// TIA Portal project "Project2" (V16)

(* hardware
DEVICE "S7-1200 station_1"  S7-1200 Station
   slot 0: "Rack_0"  S7-1200 Rack  Rack  V1.0
   slot 1: "PLC_1"  CPU 1212C AC/DC/Rly  6ES7 212-1BE40-0XB0  V4.4
*)

// ===== PLC "PLC_1"  CPU 1212C AC/DC/Rly =====

VAR_GLOBAL   // PLC tag table "Default tag table"
   "START" AT %I0.1 : Bool;
   "STOP" AT %I0.2 : Bool;
   "MOTOR1" AT %Q0.0 : Bool;
   "MOTOR2" AT %Q0.1 : Bool;
   "MOTOR3" AT %Q0.2 : Bool;
   "Tag_1" AT %M0.0 : Bool;
   "Tag_2" AT %M0.1 : Bool;
   "Tag_3" AT %M0.2 : Bool;
   "Tag_4" AT %M0.3 : Bool;
END_VAR

// folder: System blocks/Program resources

DATA_BLOCK "TIMER1"   // DB1
{ S7_Optimized_Access := 'TRUE' }
AUTHOR : Simatic
FAMILY : IEC
NAME : IEC_TMR
VERSION : 1.0
// stored: InstanceOfName IEC_TIMER
"IEC_TIMER"
BEGIN
END_DATA_BLOCK

DATA_BLOCK "TIMER2"   // DB2
{ S7_Optimized_Access := 'TRUE' }
AUTHOR : Simatic
FAMILY : IEC
NAME : IEC_TMR
VERSION : 1.0
// stored: InstanceOfName IEC_TIMER
"IEC_TIMER"
BEGIN
END_DATA_BLOCK

// folder: (top level)

ORGANIZATION_BLOCK "Main"   // OB1, LAD, ProgramCycle
TITLE = "Main Program Sweep (Cycle)"
{ S7_Optimized_Access := 'TRUE' }
VERSION : 0.1
   VAR_INPUT
      Initial_Call : Bool;   // Initial call of this OB
      Remanence : Bool;   // =True, if remanent data are available
   END_VAR
   VAR_TEMP   // added for the SCL form of the ladder/FBD networks
      _w1 : Bool;
   END_VAR
BEGIN

REGION Network 1
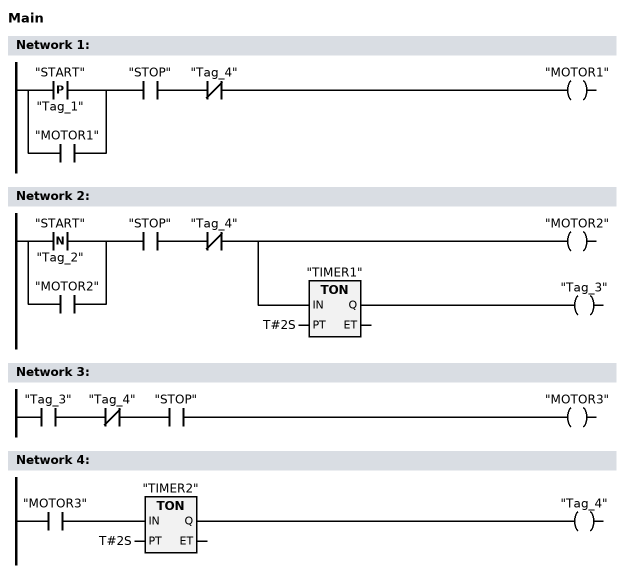
   RUNG wire#powerrail
      P_Contact(operand := "START", bit := "Tag_1")
      wire#w1
      Contact( "STOP" )
      I_Contact( "Tag_4" )
      Coil( "MOTOR1" )
   END_RUNG
   RUNG wire#powerrail
      Contact( "MOTOR1" )
   END_RUNG wire#w1
   // the same network as SCL:
   #_w1 := "START" AND NOT "Tag_1";   // rising edge of "START"
   "Tag_1" := "START";
   "MOTOR1" := (#_w1 OR "MOTOR1") AND "STOP" AND NOT "Tag_4";
END_REGION

REGION Network 2
   #_w1 := NOT "START" AND "Tag_2";   // falling edge of "START"
   "Tag_2" := "START";
   "MOTOR2" := (#_w1 OR "MOTOR2") AND "STOP" AND NOT "Tag_4";
   "TIMER1".TON(IN := "MOTOR2", PT := T#2S);
   "Tag_3" := "TIMER1".Q;
END_REGION

REGION Network 3
   RUNG wire#powerrail
      Contact( "Tag_3" )
      I_Contact( "Tag_4" )
      Contact( "STOP" )
      Coil( "MOTOR3" )
   END_RUNG
   // the same network as SCL:
   "MOTOR3" := "Tag_3" AND NOT "Tag_4" AND "STOP";
END_REGION

REGION Network 4
   "TIMER2".TON(IN := "MOTOR3", PT := T#2S);
   "Tag_4" := "TIMER2".Q;
END_REGION
END_ORGANIZATION_BLOCK